// values integer
      L     #EventObject_25; // event-Nr
      T     "SSA_LOG_Value_Queue".Input.Para_0010;
      L     2; // object-state going
      T     "SSA_LOG_Value_Queue".Input.Para_0011;
      L     0; // number additional param
      T     "SSA_LOG_Value_Queue".Input.Para_0012;
// cont log-messages
      L     "SSA_LOG_Value_Queue".Input.Para_0099; // message counter
      L     1;
      +I    ;
      T     "SSA_LOG_Value_Queue".Input.Para_0099; // message counter

// Transform Basic Time to Local Time
//      CALL  "BT_LT"
//       BT     :="DB Prozesszeit".Arbeitsbereich.dt1
//       WS_DAT :="RegelDB"
//       RET_VAL:=MW218
//       LT     :="RegelDB".LocalTime
// put timestamp into message
      CALL "SYS_Copy_DBtoDB" (
           DBSource                 := 1013,
           ByteSource               := 18,
           DBDest                   := 1005,
           ByteDest                 := 462,
           NoOfByte                 := 8,
           Fault                    := M    210.0);
///
      CALL "SSA_MH_LogEntry_ActValue" (
           DBNumber                 := 1005);

E060: NOP   0;
///
// Ereignis 26  Kommt
      U     #EREIGNISBIT_26;
      FP    #Ereignis_26.FP_Kommt;
      SPBN  E061;
// header
      L     #MessageType;
      T     "SSA_LOG_Value_Queue".Input.Header.SecType; // type
      L     #MessageFormat;
      T     "SSA_LOG_Value_Queue".Input.Header.Format; // format
      L     #JobNumber;
      T     "SSA_LOG_Value_Queue".Input.Para_0005;
      L     #processMinute;
      T     "SSA_LOG_Value_Queue".Input.Para_0007;
      L     #StepNumber;
      T     "SSA_LOG_Value_Queue".Input.Para_0008;
      L     #StepTimeMin;
      T     "SSA_LOG_Value_Queue".Input.Para_0009;

// values integer
      L     #EventObject_26; // event-Nr
      T     "SSA_LOG_Value_Queue".Input.Para_0010;
      L     1; // object-state coming
      T     "SSA_LOG_Value_Queue".Input.Para_0011;
      L     0; // number additional param
      T     "SSA_LOG_Value_Queue".Input.Para_0012;
// cont log-messages
      L     "SSA_LOG_Value_Queue".Input.Para_0099; // message counter
      L     1;
      +I    ;
      T     "SSA_LOG_Value_Queue".Input.Para_0099; // message counter

// Transform Basic Time to Local Time
//      CALL  "BT_LT"
//       BT     :="DB Prozesszeit".Arbeitsbereich.dt1
//       WS_DAT :="RegelDB"
//       RET_VAL:=MW218
//       LT     :="RegelDB".LocalTime
// put timestamp into message
      CALL "SYS_Copy_DBtoDB" (
           DBSource                 := 1013,
           ByteSource               := 18,
           DBDest                   := 1005,
           ByteDest                 := 462,
           NoOfByte                 := 8,
           Fault                    := M    210.0);
///
      CALL "SSA_MH_LogEntry_ActValue" (
           DBNumber                 := 1005);

E061: NOP   0;
///
// Ereignis 26  Geht
      U     #EREIGNISBIT_26;
      FN    #Ereignis_26.FN_Geht;
      SPBN  E062;
// header
      L     #MessageType;
      T     "SSA_LOG_Value_Queue".Input.Header.SecType; // type
      L     #MessageFormat;
      T     "SSA_LOG_Value_Queue".Input.Header.Format; // format
      L     #JobNumber;
      T     "SSA_LOG_Value_Queue".Input.Para_0005;
      L     #processMinute;
      T     "SSA_LOG_Value_Queue".Input.Para_0007;
      L     #StepNumber;
      T     "SSA_LOG_Value_Queue".Input.Para_0008;
      L     #StepTimeMin;
      T     "SSA_LOG_Value_Queue".Input.Para_0009;

// values integer
      L     #EventObject_26; // event-Nr
      T     "SSA_LOG_Value_Queue".Input.Para_0010;
      L     2; // object-state going
      T     "SSA_LOG_Value_Queue".Input.Para_0011;
      L     0; // number additional param
      T     "SSA_LOG_Value_Queue".Input.Para_0012;
// cont log-messages
      L     "SSA_LOG_Value_Queue".Input.Para_0099; // message counter
      L     1;
      +I    ;
      T     "SSA_LOG_Value_Queue".Input.Para_0099; // message counter

// Transform Basic Time to Local Time
//      CALL  "BT_LT"
//       BT     :="DB Prozesszeit".Arbeitsbereich.dt1
//       WS_DAT :="RegelDB"
//       RET_VAL:=MW218
//       LT     :="RegelDB".LocalTime
// put timestamp into message
      CALL "SYS_Copy_DBtoDB" (
           DBSource                 := 1013,
           ByteSource               := 18,
           DBDest                   := 1005,
           ByteDest                 := 462,
           NoOfByte                 := 8,
           Fault                    := M    210.0);
///
      CALL "SSA_MH_LogEntry_ActValue" (
           DBNumber                 := 1005);

E062: NOP   0;
///
// Ereignis 27  Kommt
      U     #EREIGNISBIT_27;
      FP    #Ereignis_27.FP_Kommt;
      SPBN  E063;
/// header
      L     #MessageType;
      T     "SSA_LOG_Value_Queue".Input.Header.SecType; // type
      L     #MessageFormat;
      T     "SSA_LOG_Value_Queue".Input.Header.Format; // format
      L     #JobNumber;
      T     "SSA_LOG_Value_Queue".Input.Para_0005;
      L     #processMinute;
      T     "SSA_LOG_Value_Queue".Input.Para_0007;
      L     #StepNumber;
      T     "SSA_LOG_Value_Queue".Input.Para_0008;
      L     #StepTimeMin;
      T     "SSA_LOG_Value_Queue".Input.Para_0009;

// values integer
      L     #EventObject_27; // event-Nr
      T     "SSA_LOG_Value_Queue".Input.Para_0010;
      L     1; // object-state coming
      T     "SSA_LOG_Value_Queue".Input.Para_0011;
      L     0; // number additional param
      T     "SSA_LOG_Value_Queue".Input.Para_0012;
// cont log-messages
      L     "SSA_LOG_Value_Queue".Input.Para_0099; // message counter
      L     1;
      +I    ;
      T     "SSA_LOG_Value_Queue".Input.Para_0099; // message counter

// Transform Basic Time to Local Time
//      CALL  "BT_LT"
//       BT     :="DB Prozesszeit".Arbeitsbereich.dt1
//       WS_DAT :="RegelDB"
//       RET_VAL:=MW218
//       LT     :="RegelDB".LocalTime
// put timestamp into message
      CALL "SYS_Copy_DBtoDB" (
           DBSource                 := 1013,
           ByteSource               := 18,
           DBDest                   := 1005,
           ByteDest                 := 462,
           NoOfByte                 := 8,
           Fault                    := M    210.0);
///
      CALL "SSA_MH_LogEntry_ActValue" (
           DBNumber                 := 1005);

E063: NOP   0;
///
// Ereignis 27  Geht
      U     #EREIGNISBIT_27;
      FN    #Ereignis_27.FN_Geht;
      SPBN  E064;
// header
      L     #MessageType;
      T     "SSA_LOG_Value_Queue".Input.Header.SecType; // type
      L     #MessageFormat;
      T     "SSA_LOG_Value_Queue".Input.Header.Format; // format
      L     #JobNumber;
      T     "SSA_LOG_Value_Queue".Input.Para_0005;
      L     #processMinute;
      T     "SSA_LOG_Value_Queue".Input.Para_0007;
      L     #StepNumber;
      T     "SSA_LOG_Value_Queue".Input.Para_0008;
      L     #StepTimeMin;
      T     "SSA_LOG_Value_Queue".Input.Para_0009;

// values integer
      L     #EventObject_27; // event-Nr
      T     "SSA_LOG_Value_Queue".Input.Para_0010;
      L     2; // object-state going
      T     "SSA_LOG_Value_Queue".Input.Para_0011;
      L     0; // number additional param
      T     "SSA_LOG_Value_Queue".Input.Para_0012;
// cont log-messages
      L     "SSA_LOG_Value_Queue".Input.Para_0099; // message counter
      L     1;
      +I    ;
      T     "SSA_LOG_Value_Queue".Input.Para_0099; // message counter

// Transform Basic Time to Local Time
//      CALL  "BT_LT"
//       BT     :="DB Prozesszeit".Arbeitsbereich.dt1
//       WS_DAT :="RegelDB"
//       RET_VAL:=MW218
//       LT     :="RegelDB".LocalTime
// put timestamp into message
      CALL "SYS_Copy_DBtoDB" (
           DBSource                 := 1013,
           ByteSource               := 18,
           DBDest                   := 1005,
           ByteDest                 := 462,
           NoOfByte                 := 8,
           Fault                    := M    210.0);
///
      CALL "SSA_MH_LogEntry_ActValue" (
           DBNumber                 := 1005);

E064: NOP   0;
///
// Ereignis 28  Kommt
      U     #EREIGNISBIT_28;
      FP    #Ereignis_28.FP_Kommt;
      SPBN  E065;
// header
      L     #MessageType;
      T     "SSA_LOG_Value_Queue".Input.Header.SecType; // type
      L     #MessageFormat;
      T     "SSA_LOG_Value_Queue".Input.Header.Format; // format
      L     #JobNumber;
      T     "SSA_LOG_Value_Queue".Input.Para_0005;
      L     #processMinute;
      T     "SSA_LOG_Value_Queue".Input.Para_0007;
      L     #StepNumber;
      T     "SSA_LOG_Value_Queue".Input.Para_0008;
      L     #StepTimeMin;
      T     "SSA_LOG_Value_Queue".Input.Para_0009;

// values integer
      L     #EventObject_28; // event-Nr
      T     "SSA_LOG_Value_Queue".Input.Para_0010;
      L     1; // object-state coming
      T     "SSA_LOG_Value_Queue".Input.Para_0011;
      L     0; // number additional param
      T     "SSA_LOG_Value_Queue".Input.Para_0012;
// cont log-messages
      L     "SSA_LOG_Value_Queue".Input.Para_0099; // message counter
      L     1;
      +I    ;
      T     "SSA_LOG_Value_Queue".Input.Para_0099; // message counter

// Transform Basic Time to Local Time
//      CALL  "BT_LT"
//       BT     :="DB Prozesszeit".Arbeitsbereich.dt1
//       WS_DAT :="RegelDB"
//       RET_VAL:=MW218
//       LT     :="RegelDB".LocalTime
// put timestamp into message
      CALL "SYS_Copy_DBtoDB" (
           DBSource                 := 1013,
           ByteSource               := 18,
           DBDest                   := 1005,
           ByteDest                 := 462,
           NoOfByte                 := 8,
           Fault                    := M    210.0);
///
      CALL "SSA_MH_LogEntry_ActValue" (
           DBNumber                 := 1005);

E065: NOP   0;
///
// Ereignis 28  Geht
      U     #EREIGNISBIT_28;
      FN    #Ereignis_28.FN_Geht;
      SPBN  E066;
// header
      L     #MessageType;
      T     "SSA_LOG_Value_Queue".Input.Header.SecType; // type
      L     #MessageFormat;
      T     "SSA_LOG_Value_Queue".Input.Header.Format; // format
      L     #JobNumber;
      T     "SSA_LOG_Value_Queue".Input.Para_0005;
      L     #processMinute;
      T     "SSA_LOG_Value_Queue".Input.Para_0007;
      L     #StepNumber;
      T     "SSA_LOG_Value_Queue".Input.Para_0008;
      L     #StepTimeMin;
      T     "SSA_LOG_Value_Queue".Input.Para_0009;

// values integer
      L     #EventObject_28; // event-Nr
      T     "SSA_LOG_Value_Queue".Input.Para_0010;
      L     2; // object-state going
      T     "SSA_LOG_Value_Queue".Input.Para_0011;
      L     0; // number additional param
      T     "SSA_LOG_Value_Queue".Input.Para_0012;
// cont log-messages
      L     "SSA_LOG_Value_Queue".Input.Para_0099; // message counter
      L     1;
      +I    ;
      T     "SSA_LOG_Value_Queue".Input.Para_0099; // message counter

// Transform Basic Time to Local Time
//      CALL  "BT_LT"
//       BT     :="DB Prozesszeit".Arbeitsbereich.dt1
//       WS_DAT :="RegelDB"
//       RET_VAL:=MW218
//       LT     :="RegelDB".LocalTime
// put timestamp into message
      CALL "SYS_Copy_DBtoDB" (
           DBSource                 := 1013,
           ByteSource               := 18,
           DBDest                   := 1005,
           ByteDest                 := 462,
           NoOfByte                 := 8,
           Fault                    := M    210.0);
///
      CALL "SSA_MH_LogEntry_ActValue" (
           DBNumber                 := 1005);

E066: NOP   0;
///
// Ereignis 29  Kommt
      U     #EREIGNISBIT_29;
      FP    #Ereignis_29.FP_Kommt;
      SPBN  E067;
// header
      L     #MessageType;
      T     "SSA_LOG_Value_Queue".Input.Header.SecType; // type
      L     #MessageFormat;
      T     "SSA_LOG_Value_Queue".Input.Header.Format; // format
      L     #JobNumber;
      T     "SSA_LOG_Value_Queue".Input.Para_0005;
      L     #processMinute;
      T     "SSA_LOG_Value_Queue".Input.Para_0007;
      L     #StepNumber;
      T     "SSA_LOG_Value_Queue".Input.Para_0008;
      L     #StepTimeMin;
      T     "SSA_LOG_Value_Queue".Input.Para_0009;

// values integer
      L     #EventObject_29; // event-Nr
      T     "SSA_LOG_Value_Queue".Input.Para_0010;
      L     1; // object-state coming
      T     "SSA_LOG_Value_Queue".Input.Para_0011;
      L     0; // number additional param
      T     "SSA_LOG_Value_Queue".Input.Para_0012;
// cont log-messages
      L     "SSA_LOG_Value_Queue".Input.Para_0099; // message counter
      L     1;
      +I    ;
      T     "SSA_LOG_Value_Queue".Input.Para_0099; // message counter

// Transform Basic Time to Local Time
//      CALL  "BT_LT"
//       BT     :="DB Prozesszeit".Arbeitsbereich.dt1
//       WS_DAT :="RegelDB"
//       RET_VAL:=MW218
//       LT     :="RegelDB".LocalTime
// put timestamp into message
      CALL "SYS_Copy_DBtoDB" (
           DBSource                 := 1013,
           ByteSource               := 18,
           DBDest                   := 1005,
           ByteDest                 := 462,
           NoOfByte                 := 8,
           Fault                    := M    210.0);
///
      CALL "SSA_MH_LogEntry_ActValue" (
           DBNumber                 := 1005);

E067: NOP   0;
///
// Ereignis 29  Geht
      U     #EREIGNISBIT_29;
      FN    #Ereignis_29.FN_Geht;
      SPBN  E068;
// header
      L     #MessageType;
      T     "SSA_LOG_Value_Queue".Input.Header.SecType; // type
      L     #MessageFormat;
      T     "SSA_LOG_Value_Queue".Input.Header.Format; // format
      L     #JobNumber;
      T     "SSA_LOG_Value_Queue".Input.Para_0005;
      L     #processMinute;
      T     "SSA_LOG_Value_Queue".Input.Para_0007;
      L     #StepNumber;
      T     "SSA_LOG_Value_Queue".Input.Para_0008;
      L     #StepTimeMin;
      T     "SSA_LOG_Value_Queue".Input.Para_0009;

// values integer
      L     #EventObject_29; // event-Nr
      T     "SSA_LOG_Value_Queue".Input.Para_0010;
      L     2; // object-state going
      T     "SSA_LOG_Value_Queue".Input.Para_0011;
      L     0; // number additional param
      T     "SSA_LOG_Value_Queue".Input.Para_0012;
// cont log-messages
      L     "SSA_LOG_Value_Queue".Input.Para_0099; // message counter
      L     1;
      +I    ;
      T     "SSA_LOG_Value_Queue".Input.Para_0099; // message counter

// Transform Basic Time to Local Time
//      CALL  "BT_LT"
//       BT     :="DB Prozesszeit".Arbeitsbereich.dt1
//       WS_DAT :="RegelDB"
//       RET_VAL:=MW218
//       LT     :="RegelDB".LocalTime
// put timestamp into message
      CALL "SYS_Copy_DBtoDB" (
           DBSource                 := 1013,
           ByteSource               := 18,
           DBDest                   := 1005,
           ByteDest                 := 462,
           NoOfByte                 := 8,
           Fault                    := M    210.0);
///
      CALL "SSA_MH_LogEntry_ActValue" (
           DBNumber                 := 1005);

E068: NOP   0;
///
// Ereignis 30  Kommt
      U     #EREIGNISBIT_30;
      FP    #Ereignis_30.FP_Kommt;
      SPBN  E069;
// header
      L     #MessageType;
      T     "SSA_LOG_Value_Queue".Input.Header.SecType; // type
      L     #MessageFormat;
      T     "SSA_LOG_Value_Queue".Input.Header.Format; // format
      L     #JobNumber;
      T     "SSA_LOG_Value_Queue".Input.Para_0005;
      L     #processMinute;
      T     "SSA_LOG_Value_Queue".Input.Para_0007;
      L     #StepNumber;
      T     "SSA_LOG_Value_Queue".Input.Para_0008;
      L     #StepTimeMin;
      T     "SSA_LOG_Value_Queue".Input.Para_0009;

// values integer
      L     #EventObject_30; // event-Nr
      T     "SSA_LOG_Value_Queue".Input.Para_0010;
      L     1; // object-state coming
      T     "SSA_LOG_Value_Queue".Input.Para_0011;
      L     0; // number additional param
      T     "SSA_LOG_Value_Queue".Input.Para_0012;
// cont log-messages
      L     "SSA_LOG_Value_Queue".Input.Para_0099; // message counter
      L     1;
      +I    ;
      T     "SSA_LOG_Value_Queue".Input.Para_0099; // message counter

// Transform Basic Time to Local Time
//      CALL  "BT_LT"
//       BT     :="DB Prozesszeit".Arbeitsbereich.dt1
//       WS_DAT :="RegelDB"
//       RET_VAL:=MW218
//       LT     :="RegelDB".LocalTime
// put timestamp into message
      CALL "SYS_Copy_DBtoDB" (
           DBSource                 := 1013,
           ByteSource               := 18,
           DBDest                   := 1005,
           ByteDest                 := 462,
           NoOfByte                 := 8,
           Fault                    := M    210.0);
///
      CALL "SSA_MH_LogEntry_ActValue" (
           DBNumber                 := 1005);

E069: NOP   0;
///
// Ereignis 30  Geht
      U     #EREIGNISBIT_30;
      FN    #Ereignis_30.FN_Geht;
      SPBN  E070;
// header
      L     #MessageType;
      T     "SSA_LOG_Value_Queue".Input.Header.SecType; // type
      L     #MessageFormat;
      T     "SSA_LOG_Value_Queue".Input.Header.Format; // format
      L     #JobNumber;
      T     "SSA_LOG_Value_Queue".Input.Para_0005;
      L     #processMinute;
      T     "SSA_LOG_Value_Queue".Input.Para_0007;
      L     #StepNumber;
      T     "SSA_LOG_Value_Queue".Input.Para_0008;
      L     #StepTimeMin;
      T     "SSA_LOG_Value_Queue".Input.Para_0009;

// values integer
      L     #EventObject_30; // event-Nr
      T     "SSA_LOG_Value_Queue".Input.Para_0010;
      L     2; // object-state going
      T     "SSA_LOG_Value_Queue".Input.Para_0011;
      L     0; // number additional param
      T     "SSA_LOG_Value_Queue".Input.Para_0012;
// cont log-messages
      L     "SSA_LOG_Value_Queue".Input.Para_0099; // message counter
      L     1;
      +I    ;
      T     "SSA_LOG_Value_Queue".Input.Para_0099; // message counter

// Transform Basic Time to Local Time
//      CALL  "BT_LT"
//       BT     :="DB Prozesszeit".Arbeitsbereich.dt1
//       WS_DAT :="RegelDB"
//       RET_VAL:=MW218
//       LT     :="RegelDB".LocalTime
// put timestamp into message
      CALL "SYS_Copy_DBtoDB" (
           DBSource                 := 1013,
           ByteSource               := 18,
           DBDest                   := 1005,
           ByteDest                 := 462,
           NoOfByte                 := 8,
           Fault                    := M    210.0);
///
      CALL "SSA_MH_LogEntry_ActValue" (
           DBNumber                 := 1005);

E070: NOP   0;
///

NETWORK
TITLE =create events for batchprotokoll
//event Nr. 121 - 130 are  events in job-protocol
///
// Ereignis 31  Kommt
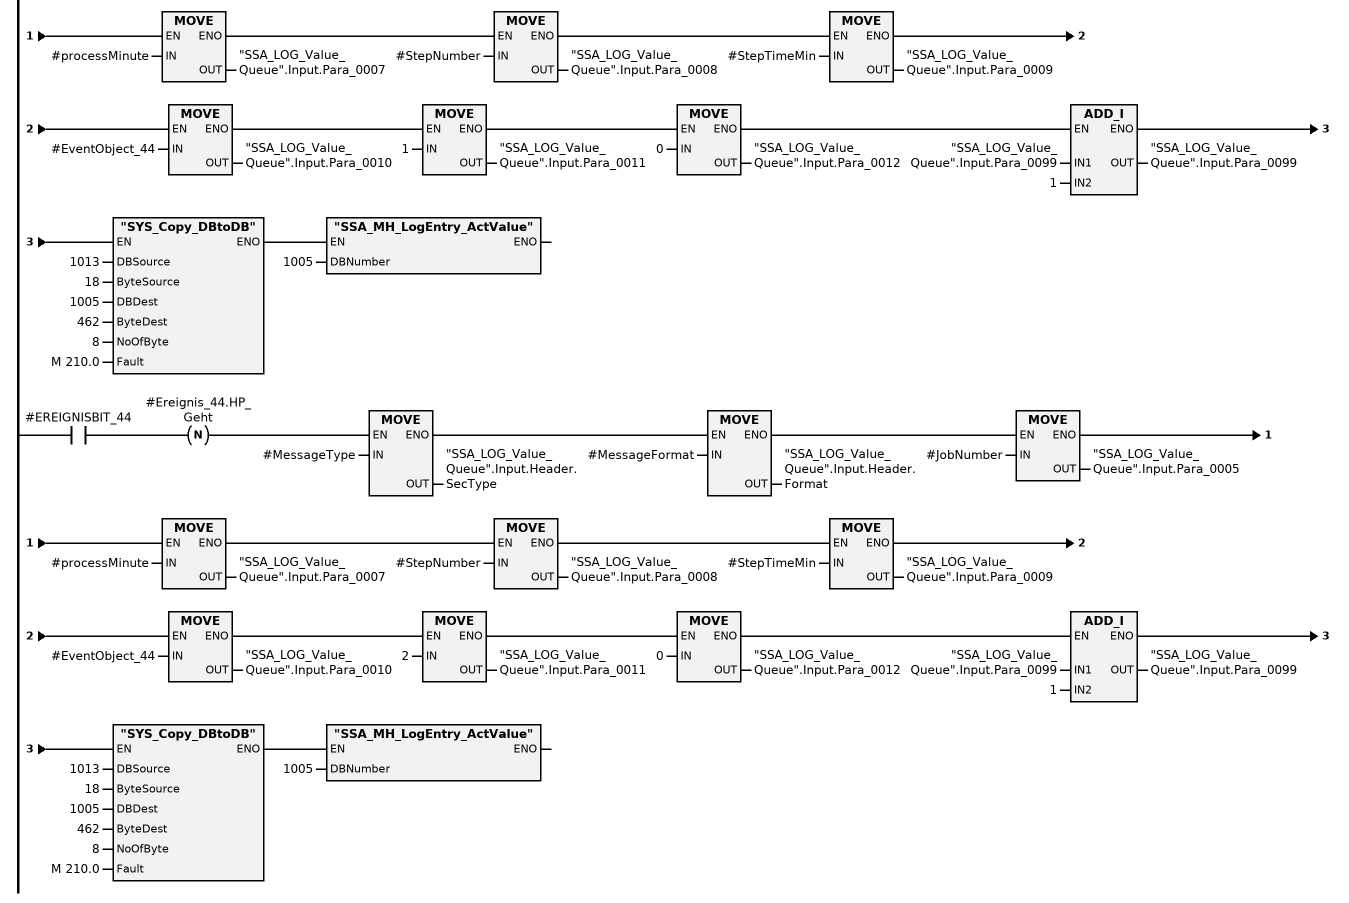
      U     #EREIGNISBIT_31;
      FP    #Ereignis_31.FP_Kommt;
      SPBN  E071;
// header
      L     #MessageType;
      T     "SSA_LOG_Value_Queue".Input.Header.SecType; // type
      L     #MessageFormat;
      T     "SSA_LOG_Value_Queue".Input.Header.Format; // format
      L     #JobNumber;
      T     "SSA_LOG_Value_Queue".Input.Para_0005;
      L     #processMinute;
      T     "SSA_LOG_Value_Queue".Input.Para_0007;
      L     #StepNumber;
      T     "SSA_LOG_Value_Queue".Input.Para_0008;
      L     #StepTimeMin;
      T     "SSA_LOG_Value_Queue".Input.Para_0009;

// values integer
      L     #EventObject_31; // event-Nr
      T     "SSA_LOG_Value_Queue".Input.Para_0010;
      L     1; // object-state coming
      T     "SSA_LOG_Value_Queue".Input.Para_0011;
      L     0; // number additional param
      T     "SSA_LOG_Value_Queue".Input.Para_0012;
// cont log-messages
      L     "SSA_LOG_Value_Queue".Input.Para_0099; // message counter
      L     1;
      +I    ;
      T     "SSA_LOG_Value_Queue".Input.Para_0099; // message counter

// Transform Basic Time to Local Time
//      CALL  "BT_LT"
//       BT     :="DB Prozesszeit".Arbeitsbereich.dt1
//       WS_DAT :="RegelDB"
//       RET_VAL:=MW218
//       LT     :="RegelDB".LocalTime
// put timestamp into message
      CALL "SYS_Copy_DBtoDB" (
           DBSource                 := 1013,
           ByteSource               := 18,
           DBDest                   := 1005,
           ByteDest                 := 462,
           NoOfByte                 := 8,
           Fault                    := M    210.0);
///
      CALL "SSA_MH_LogEntry_ActValue" (
           DBNumber                 := 1005);
E071: NOP   0;
///
// Ereignis 31  Geht
      U     #EREIGNISBIT_31;
      FN    #Ereignis_31.FN_Geht;
      SPBN  E072;
// header
      L     #MessageType;
      T     "SSA_LOG_Value_Queue".Input.Header.SecType; // type
      L     #MessageFormat;
      T     "SSA_LOG_Value_Queue".Input.Header.Format; // format
      L     #JobNumber;
      T     "SSA_LOG_Value_Queue".Input.Para_0005;
      L     #processMinute;
      T     "SSA_LOG_Value_Queue".Input.Para_0007;
      L     #StepNumber;
      T     "SSA_LOG_Value_Queue".Input.Para_0008;
      L     #StepTimeMin;
      T     "SSA_LOG_Value_Queue".Input.Para_0009;

// values integer
      L     #EventObject_31; // event-Nr
      T     "SSA_LOG_Value_Queue".Input.Para_0010;
      L     2; // object-state going
      T     "SSA_LOG_Value_Queue".Input.Para_0011;
      L     0; // number additional param
      T     "SSA_LOG_Value_Queue".Input.Para_0012;
// cont log-messages
      L     "SSA_LOG_Value_Queue".Input.Para_0099; // message counter
      L     1;
      +I    ;
      T     "SSA_LOG_Value_Queue".Input.Para_0099; // message counter

// Transform Basic Time to Local Time
//      CALL  "BT_LT"
//       BT     :="DB Prozesszeit".Arbeitsbereich.dt1
//       WS_DAT :="RegelDB"
//       RET_VAL:=MW218
//       LT     :="RegelDB".LocalTime
// put timestamp into message
      CALL "SYS_Copy_DBtoDB" (
           DBSource                 := 1013,
           ByteSource               := 18,
           DBDest                   := 1005,
           ByteDest                 := 462,
           NoOfByte                 := 8,
           Fault                    := M    210.0);
///
      CALL "SSA_MH_LogEntry_ActValue" (
           DBNumber                 := 1005);

E072: NOP   0;
///
// Ereignis 32  Kommt
      U     #EREIGNISBIT_32;
      FP    #Ereignis_32.FP_Kommt;
      SPBN  E073;
// header
      L     #MessageType;
      T     "SSA_LOG_Value_Queue".Input.Header.SecType; // type
      L     #MessageFormat;
      T     "SSA_LOG_Value_Queue".Input.Header.Format; // format
      L     #JobNumber;
      T     "SSA_LOG_Value_Queue".Input.Para_0005;
      L     #processMinute;
      T     "SSA_LOG_Value_Queue".Input.Para_0007;
      L     #StepNumber;
      T     "SSA_LOG_Value_Queue".Input.Para_0008;
      L     #StepTimeMin;
      T     "SSA_LOG_Value_Queue".Input.Para_0009;

// values integer
      L     #EventObject_32; // event-Nr
      T     "SSA_LOG_Value_Queue".Input.Para_0010;
      L     1; // object-state coming
      T     "SSA_LOG_Value_Queue".Input.Para_0011;
      L     0; // number additional param
      T     "SSA_LOG_Value_Queue".Input.Para_0012;
// cont log-messages
      L     "SSA_LOG_Value_Queue".Input.Para_0099; // message counter
      L     1;
      +I    ;
      T     "SSA_LOG_Value_Queue".Input.Para_0099; // message counter

// Transform Basic Time to Local Time
//      CALL  "BT_LT"
//       BT     :="DB Prozesszeit".Arbeitsbereich.dt1
//       WS_DAT :="RegelDB"
//       RET_VAL:=MW218
//       LT     :="RegelDB".LocalTime
// put timestamp into message
      CALL "SYS_Copy_DBtoDB" (
           DBSource                 := 1013,
           ByteSource               := 18,
           DBDest                   := 1005,
           ByteDest                 := 462,
           NoOfByte                 := 8,
           Fault                    := M    210.0);
///
      CALL "SSA_MH_LogEntry_ActValue" (
           DBNumber                 := 1005);

E073: NOP   0;
///
// Ereignis 32  Geht
      U     #EREIGNISBIT_32;
      FN    #Ereignis_32.FN_Geht;
      SPBN  E074;
// header
      L     #MessageType;
      T     "SSA_LOG_Value_Queue".Input.Header.SecType; // type
      L     #MessageFormat;
      T     "SSA_LOG_Value_Queue".Input.Header.Format; // format
      L     #JobNumber;
      T     "SSA_LOG_Value_Queue".Input.Para_0005;
      L     #processMinute;
      T     "SSA_LOG_Value_Queue".Input.Para_0007;
      L     #StepNumber;
      T     "SSA_LOG_Value_Queue".Input.Para_0008;
      L     #StepTimeMin;
      T     "SSA_LOG_Value_Queue".Input.Para_0009;

// values integer
      L     #EventObject_32; // event-Nr
      T     "SSA_LOG_Value_Queue".Input.Para_0010;
      L     2; // object-state going
      T     "SSA_LOG_Value_Queue".Input.Para_0011;
      L     0; // number additional param
      T     "SSA_LOG_Value_Queue".Input.Para_0012;
// cont log-messages
      L     "SSA_LOG_Value_Queue".Input.Para_0099; // message counter
      L     1;
      +I    ;
      T     "SSA_LOG_Value_Queue".Input.Para_0099; // message counter

// Transform Basic Time to Local Time
//      CALL  "BT_LT"
//       BT     :="DB Prozesszeit".Arbeitsbereich.dt1
//       WS_DAT :="RegelDB"
//       RET_VAL:=MW218
//       LT     :="RegelDB".LocalTime
// put timestamp into message
      CALL "SYS_Copy_DBtoDB" (
           DBSource                 := 1013,
           ByteSource               := 18,
           DBDest                   := 1005,
           ByteDest                 := 462,
           NoOfByte                 := 8,
           Fault                    := M    210.0);
///
      CALL "SSA_MH_LogEntry_ActValue" (
           DBNumber                 := 1005);

E074: NOP   0;
///
// Ereignis 33  Kommt
      U     #EREIGNISBIT_33;
      FP    #Ereignis_33.FP_Kommt;
      SPBN  E075;
// header
      L     #MessageType;
      T     "SSA_LOG_Value_Queue".Input.Header.SecType; // type
      L     #MessageFormat;
      T     "SSA_LOG_Value_Queue".Input.Header.Format; // format
      L     #JobNumber;
      T     "SSA_LOG_Value_Queue".Input.Para_0005;
      L     #processMinute;
      T     "SSA_LOG_Value_Queue".Input.Para_0007;
      L     #StepNumber;
      T     "SSA_LOG_Value_Queue".Input.Para_0008;
      L     #StepTimeMin;
      T     "SSA_LOG_Value_Queue".Input.Para_0009;

// values integer
      L     #EventObject_33; // event-Nr
      T     "SSA_LOG_Value_Queue".Input.Para_0010;
      L     1; // object-state coming
      T     "SSA_LOG_Value_Queue".Input.Para_0011;
      L     0; // number additional param
      T     "SSA_LOG_Value_Queue".Input.Para_0012;
// cont log-messages
      L     "SSA_LOG_Value_Queue".Input.Para_0099; // message counter
      L     1;
      +I    ;
      T     "SSA_LOG_Value_Queue".Input.Para_0099; // message counter

// Transform Basic Time to Local Time
//      CALL  "BT_LT"
//       BT     :="DB Prozesszeit".Arbeitsbereich.dt1
//       WS_DAT :="RegelDB"
//       RET_VAL:=MW218
//       LT     :="RegelDB".LocalTime
// put timestamp into message
      CALL "SYS_Copy_DBtoDB" (
           DBSource                 := 1013,
           ByteSource               := 18,
           DBDest                   := 1005,
           ByteDest                 := 462,
           NoOfByte                 := 8,
           Fault                    := M    210.0);
///
      CALL "SSA_MH_LogEntry_ActValue" (
           DBNumber                 := 1005);

E075: NOP   0;
///
// Ereignis 33  Geht
      U     #EREIGNISBIT_33;
      FN    #Ereignis_33.FN_Geht;
      SPBN  E076;
// header
      L     #MessageType;
      T     "SSA_LOG_Value_Queue".Input.Header.SecType; // type
      L     #MessageFormat;
      T     "SSA_LOG_Value_Queue".Input.Header.Format; // format
      L     #JobNumber;
      T     "SSA_LOG_Value_Queue".Input.Para_0005;
      L     #processMinute;
      T     "SSA_LOG_Value_Queue".Input.Para_0007;
      L     #StepNumber;
      T     "SSA_LOG_Value_Queue".Input.Para_0008;
      L     #StepTimeMin;
      T     "SSA_LOG_Value_Queue".Input.Para_0009;

// values integer
      L     #EventObject_33; // event-Nr
      T     "SSA_LOG_Value_Queue".Input.Para_0010;
      L     2; // object-state going
      T     "SSA_LOG_Value_Queue".Input.Para_0011;
      L     0; // number additional param
      T     "SSA_LOG_Value_Queue".Input.Para_0012;
// cont log-messages
      L     "SSA_LOG_Value_Queue".Input.Para_0099; // message counter
      L     1;
      +I    ;
      T     "SSA_LOG_Value_Queue".Input.Para_0099; // message counter

// Transform Basic Time to Local Time
//      CALL  "BT_LT"
//       BT     :="DB Prozesszeit".Arbeitsbereich.dt1
//       WS_DAT :="RegelDB"
//       RET_VAL:=MW218
//       LT     :="RegelDB".LocalTime
// put timestamp into message
      CALL "SYS_Copy_DBtoDB" (
           DBSource                 := 1013,
           ByteSource               := 18,
           DBDest                   := 1005,
           ByteDest                 := 462,
           NoOfByte                 := 8,
           Fault                    := M    210.0);
///
      CALL "SSA_MH_LogEntry_ActValue" (
           DBNumber                 := 1005);

E076: NOP   0;
///
// Ereignis 34  Kommt
      U     #EREIGNISBIT_34;
      FP    #Ereignis_34.FP_Kommt;
      SPBN  E077;
// header
      L     #MessageType;
      T     "SSA_LOG_Value_Queue".Input.Header.SecType; // type
      L     #MessageFormat;
      T     "SSA_LOG_Value_Queue".Input.Header.Format; // format
      L     #JobNumber;
      T     "SSA_LOG_Value_Queue".Input.Para_0005;
      L     #processMinute;
      T     "SSA_LOG_Value_Queue".Input.Para_0007;
      L     #StepNumber;
      T     "SSA_LOG_Value_Queue".Input.Para_0008;
      L     #StepTimeMin;
      T     "SSA_LOG_Value_Queue".Input.Para_0009;

// values integer
      L     #EventObject_34; // event-Nr
      T     "SSA_LOG_Value_Queue".Input.Para_0010;
      L     1; // object-state coming
      T     "SSA_LOG_Value_Queue".Input.Para_0011;
      L     0; // number additional param
      T     "SSA_LOG_Value_Queue".Input.Para_0012;
// cont log-messages
      L     "SSA_LOG_Value_Queue".Input.Para_0099; // message counter
      L     1;
      +I    ;
      T     "SSA_LOG_Value_Queue".Input.Para_0099; // message counter

// Transform Basic Time to Local Time
//      CALL  "BT_LT"
//       BT     :="DB Prozesszeit".Arbeitsbereich.dt1
//       WS_DAT :="RegelDB"
//       RET_VAL:=MW218
//       LT     :="RegelDB".LocalTime
// put timestamp into message
      CALL "SYS_Copy_DBtoDB" (
           DBSource                 := 1013,
           ByteSource               := 18,
           DBDest                   := 1005,
           ByteDest                 := 462,
           NoOfByte                 := 8,
           Fault                    := M    210.0);
///
      CALL "SSA_MH_LogEntry_ActValue" (
           DBNumber                 := 1005);

E077: NOP   0;
///
// Ereignis 34  Geht
      U     #EREIGNISBIT_34;
      FN    #Ereignis_34.FN_Geht;
      SPBN  E078;
// header
      L     #MessageType;
      T     "SSA_LOG_Value_Queue".Input.Header.SecType; // type
      L     #MessageFormat;
      T     "SSA_LOG_Value_Queue".Input.Header.Format; // format
      L     #JobNumber;
      T     "SSA_LOG_Value_Queue".Input.Para_0005;
      L     #processMinute;
      T     "SSA_LOG_Value_Queue".Input.Para_0007;
      L     #StepNumber;
      T     "SSA_LOG_Value_Queue".Input.Para_0008;
      L     #StepTimeMin;
      T     "SSA_LOG_Value_Queue".Input.Para_0009;

// values integer
      L     #EventObject_34; // event-Nr
      T     "SSA_LOG_Value_Queue".Input.Para_0010;
      L     2; // object-state going
      T     "SSA_LOG_Value_Queue".Input.Para_0011;
      L     0; // number additional param
      T     "SSA_LOG_Value_Queue".Input.Para_0012;
// cont log-messages
      L     "SSA_LOG_Value_Queue".Input.Para_0099; // message counter
      L     1;
      +I    ;
      T     "SSA_LOG_Value_Queue".Input.Para_0099; // message counter

// Transform Basic Time to Local Time
//      CALL  "BT_LT"
//       BT     :="DB Prozesszeit".Arbeitsbereich.dt1
//       WS_DAT :="RegelDB"
//       RET_VAL:=MW218
//       LT     :="RegelDB".LocalTime
// put timestamp into message
      CALL "SYS_Copy_DBtoDB" (
           DBSource                 := 1013,
           ByteSource               := 18,
           DBDest                   := 1005,
           ByteDest                 := 462,
           NoOfByte                 := 8,
           Fault                    := M    210.0);
///
      CALL "SSA_MH_LogEntry_ActValue" (
           DBNumber                 := 1005);

E078: NOP   0;
///
// Ereignis 35  Kommt
      U     #EREIGNISBIT_35;
      FP    #Ereignis_35.FP_Kommt;
      SPBN  E079;
// header
      L     #MessageType;
      T     "SSA_LOG_Value_Queue".Input.Header.SecType; // type
      L     #MessageFormat;
      T     "SSA_LOG_Value_Queue".Input.Header.Format; // format
      L     #JobNumber;
      T     "SSA_LOG_Value_Queue".Input.Para_0005;
      L     #processMinute;
      T     "SSA_LOG_Value_Queue".Input.Para_0007;
      L     #StepNumber;
      T     "SSA_LOG_Value_Queue".Input.Para_0008;
      L     #StepTimeMin;
      T     "SSA_LOG_Value_Queue".Input.Para_0009;

// values integer
      L     #EventObject_35; // event-Nr
      T     "SSA_LOG_Value_Queue".Input.Para_0010;
      L     1; // object-state coming
      T     "SSA_LOG_Value_Queue".Input.Para_0011;
      L     0; // number additional param
      T     "SSA_LOG_Value_Queue".Input.Para_0012;
// cont log-messages
      L     "SSA_LOG_Value_Queue".Input.Para_0099; // message counter
      L     1;
      +I    ;
      T     "SSA_LOG_Value_Queue".Input.Para_0099; // message counter

// Transform Basic Time to Local Time
//      CALL  "BT_LT"
//       BT     :="DB Prozesszeit".Arbeitsbereich.dt1
//       WS_DAT :="RegelDB"
//       RET_VAL:=MW218
//       LT     :="RegelDB".LocalTime
// put timestamp into message
      CALL "SYS_Copy_DBtoDB" (
           DBSource                 := 1013,
           ByteSource               := 18,
           DBDest                   := 1005,
           ByteDest                 := 462,
           NoOfByte                 := 8,
           Fault                    := M    210.0);
///
      CALL "SSA_MH_LogEntry_ActValue" (
           DBNumber                 := 1005);

E079: NOP   0;
///
// Ereignis 35  Geht
      U     #EREIGNISBIT_35;
      FN    #Ereignis_35.FN_Geht;
      SPBN  E080;
// header
      L     #MessageType;
      T     "SSA_LOG_Value_Queue".Input.Header.SecType; // type
      L     #MessageFormat;
      T     "SSA_LOG_Value_Queue".Input.Header.Format; // format
      L     #JobNumber;
      T     "SSA_LOG_Value_Queue".Input.Para_0005;
      L     #processMinute;
      T     "SSA_LOG_Value_Queue".Input.Para_0007;
      L     #StepNumber;
      T     "SSA_LOG_Value_Queue".Input.Para_0008;
      L     #StepTimeMin;
      T     "SSA_LOG_Value_Queue".Input.Para_0009;

// values integer
      L     #EventObject_35; // event-Nr
      T     "SSA_LOG_Value_Queue".Input.Para_0010;
      L     2; // object-state going
      T     "SSA_LOG_Value_Queue".Input.Para_0011;
      L     0; // number additional param
      T     "SSA_LOG_Value_Queue".Input.Para_0012;
// cont log-messages
      L     "SSA_LOG_Value_Queue".Input.Para_0099; // message counter
      L     1;
      +I    ;
      T     "SSA_LOG_Value_Queue".Input.Para_0099; // message counter

// Transform Basic Time to Local Time
//      CALL  "BT_LT"
//       BT     :="DB Prozesszeit".Arbeitsbereich.dt1
//       WS_DAT :="RegelDB"
//       RET_VAL:=MW218
//       LT     :="RegelDB".LocalTime
// put timestamp into message
      CALL "SYS_Copy_DBtoDB" (
           DBSource                 := 1013,
           ByteSource               := 18,
           DBDest                   := 1005,
           ByteDest                 := 462,
           NoOfByte                 := 8,
           Fault                    := M    210.0);
///
      CALL "SSA_MH_LogEntry_ActValue" (
           DBNumber                 := 1005);

E080: NOP   0;
///
// Ereignis 36  Kommt
      U     #EREIGNISBIT_36;
      FP    #Ereignis_36.FP_Kommt;
      SPBN  E081;
// header
      L     #MessageType;
      T     "SSA_LOG_Value_Queue".Input.Header.SecType; // type
      L     #MessageFormat;
      T     "SSA_LOG_Value_Queue".Input.Header.Format; // format
      L     #JobNumber;
      T     "SSA_LOG_Value_Queue".Input.Para_0005;
      L     #processMinute;
      T     "SSA_LOG_Value_Queue".Input.Para_0007;
      L     #StepNumber;
      T     "SSA_LOG_Value_Queue".Input.Para_0008;
      L     #StepTimeMin;
      T     "SSA_LOG_Value_Queue".Input.Para_0009;

// values integer
      L     #EventObject_36; // event-Nr
      T     "SSA_LOG_Value_Queue".Input.Para_0010;
      L     1; // object-state coming
      T     "SSA_LOG_Value_Queue".Input.Para_0011;
      L     0; // number additional param
      T     "SSA_LOG_Value_Queue".Input.Para_0012;
// cont log-messages
      L     "SSA_LOG_Value_Queue".Input.Para_0099; // message counter
      L     1;
      +I    ;
      T     "SSA_LOG_Value_Queue".Input.Para_0099; // message counter

// Transform Basic Time to Local Time
//      CALL  "BT_LT"
//       BT     :="DB Prozesszeit".Arbeitsbereich.dt1
//       WS_DAT :="RegelDB"
//       RET_VAL:=MW218
//       LT     :="RegelDB".LocalTime
// put timestamp into message
      CALL "SYS_Copy_DBtoDB" (
           DBSource                 := 1013,
           ByteSource               := 18,
           DBDest                   := 1005,
           ByteDest                 := 462,
           NoOfByte                 := 8,
           Fault                    := M    210.0);
///
      CALL "SSA_MH_LogEntry_ActValue" (
           DBNumber                 := 1005);

E081: NOP   0;
///
// Ereignis 36  Geht
      U     #EREIGNISBIT_36;
      FN    #Ereignis_36.FN_Geht;
      SPBN  E082;
// header
      L     #MessageType;
      T     "SSA_LOG_Value_Queue".Input.Header.SecType; // type
      L     #MessageFormat;
      T     "SSA_LOG_Value_Queue".Input.Header.Format; // format
      L     #JobNumber;
      T     "SSA_LOG_Value_Queue".Input.Para_0005;
      L     #processMinute;
      T     "SSA_LOG_Value_Queue".Input.Para_0007;
      L     #StepNumber;
      T     "SSA_LOG_Value_Queue".Input.Para_0008;
      L     #StepTimeMin;
      T     "SSA_LOG_Value_Queue".Input.Para_0009;

// values integer
      L     #EventObject_36; // event-Nr
      T     "SSA_LOG_Value_Queue".Input.Para_0010;
      L     2; // object-state going
      T     "SSA_LOG_Value_Queue".Input.Para_0011;
      L     0; // number additional param
      T     "SSA_LOG_Value_Queue".Input.Para_0012;
// cont log-messages
      L     "SSA_LOG_Value_Queue".Input.Para_0099; // message counter
      L     1;
      +I    ;
      T     "SSA_LOG_Value_Queue".Input.Para_0099; // message counter

// Transform Basic Time to Local Time
//      CALL  "BT_LT"
//       BT     :="DB Prozesszeit".Arbeitsbereich.dt1
//       WS_DAT :="RegelDB"
//       RET_VAL:=MW218
//       LT     :="RegelDB".LocalTime
// put timestamp into message
      CALL "SYS_Copy_DBtoDB" (
           DBSource                 := 1013,
           ByteSource               := 18,
           DBDest                   := 1005,
           ByteDest                 := 462,
           NoOfByte                 := 8,
           Fault                    := M    210.0);
///
      CALL "SSA_MH_LogEntry_ActValue" (
           DBNumber                 := 1005);

E082: NOP   0;
///
// Ereignis 37  Kommt
      U     #EREIGNISBIT_37;
      FP    #Ereignis_37.FP_Kommt;
      SPBN  E083;
// header
      L     #MessageType;
      T     "SSA_LOG_Value_Queue".Input.Header.SecType; // type
      L     #MessageFormat;
      T     "SSA_LOG_Value_Queue".Input.Header.Format; // format
      L     #JobNumber;
      T     "SSA_LOG_Value_Queue".Input.Para_0005;
      L     #processMinute;
      T     "SSA_LOG_Value_Queue".Input.Para_0007;
      L     #StepNumber;
      T     "SSA_LOG_Value_Queue".Input.Para_0008;
      L     #StepTimeMin;
      T     "SSA_LOG_Value_Queue".Input.Para_0009;

// values integer
      L     #EventObject_37; // event-Nr
      T     "SSA_LOG_Value_Queue".Input.Para_0010;
      L     1; // object-state coming
      T     "SSA_LOG_Value_Queue".Input.Para_0011;
      L     0; // number additional param
      T     "SSA_LOG_Value_Queue".Input.Para_0012;
// cont log-messages
      L     "SSA_LOG_Value_Queue".Input.Para_0099; // message counter
      L     1;
      +I    ;
      T     "SSA_LOG_Value_Queue".Input.Para_0099; // message counter

// Transform Basic Time to Local Time
//      CALL  "BT_LT"
//       BT     :="DB Prozesszeit".Arbeitsbereich.dt1
//       WS_DAT :="RegelDB"
//       RET_VAL:=MW218
//       LT     :="RegelDB".LocalTime
// put timestamp into message
      CALL "SYS_Copy_DBtoDB" (
           DBSource                 := 1013,
           ByteSource               := 18,
           DBDest                   := 1005,
           ByteDest                 := 462,
           NoOfByte                 := 8,
           Fault                    := M    210.0);
///
      CALL "SSA_MH_LogEntry_ActValue" (
           DBNumber                 := 1005);

E083: NOP   0;
///
// Ereignis 37  Geht
      U     #EREIGNISBIT_37;
      FN    #Ereignis_37.FN_Geht;
      SPBN  E084;
// header
      L     #MessageType;
      T     "SSA_LOG_Value_Queue".Input.Header.SecType; // type
      L     #MessageFormat;
      T     "SSA_LOG_Value_Queue".Input.Header.Format; // format
      L     #JobNumber;
      T     "SSA_LOG_Value_Queue".Input.Para_0005;
      L     #processMinute;
      T     "SSA_LOG_Value_Queue".Input.Para_0007;
      L     #StepNumber;
      T     "SSA_LOG_Value_Queue".Input.Para_0008;
      L     #StepTimeMin;
      T     "SSA_LOG_Value_Queue".Input.Para_0009;

// values integer
      L     #EventObject_37; // event-Nr
      T     "SSA_LOG_Value_Queue".Input.Para_0010;
      L     2; // object-state going
      T     "SSA_LOG_Value_Queue".Input.Para_0011;
      L     0; // number additional param
      T     "SSA_LOG_Value_Queue".Input.Para_0012;
// cont log-messages
      L     "SSA_LOG_Value_Queue".Input.Para_0099; // message counter
      L     1;
      +I    ;
      T     "SSA_LOG_Value_Queue".Input.Para_0099; // message counter

// Transform Basic Time to Local Time
//      CALL  "BT_LT"
//       BT     :="DB Prozesszeit".Arbeitsbereich.dt1
//       WS_DAT :="RegelDB"
//       RET_VAL:=MW218
//       LT     :="RegelDB".LocalTime
// put timestamp into message
      CALL "SYS_Copy_DBtoDB" (
           DBSource                 := 1013,
           ByteSource               := 18,
           DBDest                   := 1005,
           ByteDest                 := 462,
           NoOfByte                 := 8,
           Fault                    := M    210.0);
///
      CALL "SSA_MH_LogEntry_ActValue" (
           DBNumber                 := 1005);

E084: NOP   0;
///
// Ereignis 38  Kommt
      U     #EREIGNISBIT_38;
      FP    #Ereignis_38.FP_Kommt;
      SPBN  E085;
// header
      L     #MessageType;
      T     "SSA_LOG_Value_Queue".Input.Header.SecType; // type
      L     #MessageFormat;
      T     "SSA_LOG_Value_Queue".Input.Header.Format; // format
      L     #JobNumber;
      T     "SSA_LOG_Value_Queue".Input.Para_0005;
      L     #processMinute;
      T     "SSA_LOG_Value_Queue".Input.Para_0007;
      L     #StepNumber;
      T     "SSA_LOG_Value_Queue".Input.Para_0008;
      L     #StepTimeMin;
      T     "SSA_LOG_Value_Queue".Input.Para_0009;

// values integer
      L     #EventObject_38; // event-Nr
      T     "SSA_LOG_Value_Queue".Input.Para_0010;
      L     1; // object-state coming
      T     "SSA_LOG_Value_Queue".Input.Para_0011;
      L     0; // number additional param
      T     "SSA_LOG_Value_Queue".Input.Para_0012;
// cont log-messages
      L     "SSA_LOG_Value_Queue".Input.Para_0099; // message counter
      L     1;
      +I    ;
      T     "SSA_LOG_Value_Queue".Input.Para_0099; // message counter

// Transform Basic Time to Local Time
//      CALL  "BT_LT"
//       BT     :="DB Prozesszeit".Arbeitsbereich.dt1
//       WS_DAT :="RegelDB"
//       RET_VAL:=MW218
//       LT     :="RegelDB".LocalTime
// put timestamp into message
      CALL "SYS_Copy_DBtoDB" (
           DBSource                 := 1013,
           ByteSource               := 18,
           DBDest                   := 1005,
           ByteDest                 := 462,
           NoOfByte                 := 8,
           Fault                    := M    210.0);
///
      CALL "SSA_MH_LogEntry_ActValue" (
           DBNumber                 := 1005);

E085: NOP   0;
///
// Ereignis 38  Geht
      U     #EREIGNISBIT_38;
      FN    #Ereignis_38.FN_Geht;
      SPBN  E086;
// header
      L     #MessageType;
      T     "SSA_LOG_Value_Queue".Input.Header.SecType; // type
      L     #MessageFormat;
      T     "SSA_LOG_Value_Queue".Input.Header.Format; // format
      L     #JobNumber;
      T     "SSA_LOG_Value_Queue".Input.Para_0005;
      L     #processMinute;
      T     "SSA_LOG_Value_Queue".Input.Para_0007;
      L     #StepNumber;
      T     "SSA_LOG_Value_Queue".Input.Para_0008;
      L     #StepTimeMin;
      T     "SSA_LOG_Value_Queue".Input.Para_0009;

// values integer
      L     #EventObject_38; // event-Nr
      T     "SSA_LOG_Value_Queue".Input.Para_0010;
      L     2; // object-state going
      T     "SSA_LOG_Value_Queue".Input.Para_0011;
      L     0; // number additional param
      T     "SSA_LOG_Value_Queue".Input.Para_0012;
// cont log-messages
      L     "SSA_LOG_Value_Queue".Input.Para_0099; // message counter
      L     1;
      +I    ;
      T     "SSA_LOG_Value_Queue".Input.Para_0099; // message counter

// Transform Basic Time to Local Time
//      CALL  "BT_LT"
//       BT     :="DB Prozesszeit".Arbeitsbereich.dt1
//       WS_DAT :="RegelDB"
//       RET_VAL:=MW218
//       LT     :="RegelDB".LocalTime
// put timestamp into message
      CALL "SYS_Copy_DBtoDB" (
           DBSource                 := 1013,
           ByteSource               := 18,
           DBDest                   := 1005,
           ByteDest                 := 462,
           NoOfByte                 := 8,
           Fault                    := M    210.0);
///
      CALL "SSA_MH_LogEntry_ActValue" (
           DBNumber                 := 1005);

E086: NOP   0;
///
// Ereignis 39  Kommt
      U     #EREIGNISBIT_39;
      FP    #Ereignis_39.FP_Kommt;
      SPBN  E087;
// header
      L     #MessageType;
      T     "SSA_LOG_Value_Queue".Input.Header.SecType; // type
      L     #MessageFormat;
      T     "SSA_LOG_Value_Queue".Input.Header.Format; // format
      L     #JobNumber;
      T     "SSA_LOG_Value_Queue".Input.Para_0005;
      L     #processMinute;
      T     "SSA_LOG_Value_Queue".Input.Para_0007;
      L     #StepNumber;
      T     "SSA_LOG_Value_Queue".Input.Para_0008;
      L     #StepTimeMin;
      T     "SSA_LOG_Value_Queue".Input.Para_0009;

// values integer
      L     #EventObject_39; // event-Nr
      T     "SSA_LOG_Value_Queue".Input.Para_0010;
      L     1; // object-state coming
      T     "SSA_LOG_Value_Queue".Input.Para_0011;
      L     0; // number additional param
      T     "SSA_LOG_Value_Queue".Input.Para_0012;
// cont log-messages
      L     "SSA_LOG_Value_Queue".Input.Para_0099; // message counter
      L     1;
      +I    ;
      T     "SSA_LOG_Value_Queue".Input.Para_0099; // message counter

// Transform Basic Time to Local Time
//      CALL  "BT_LT"
//       BT     :="DB Prozesszeit".Arbeitsbereich.dt1
//       WS_DAT :="RegelDB"
//       RET_VAL:=MW218
//       LT     :="RegelDB".LocalTime
// put timestamp into message
      CALL "SYS_Copy_DBtoDB" (
           DBSource                 := 1013,
           ByteSource               := 18,
           DBDest                   := 1005,
           ByteDest                 := 462,
           NoOfByte                 := 8,
           Fault                    := M    210.0);
///
      CALL "SSA_MH_LogEntry_ActValue" (
           DBNumber                 := 1005);

E087: NOP   0;
///
// Ereignis 39  Geht
      U     #EREIGNISBIT_39;
      FN    #Ereignis_39.FN_Geht;
      SPBN  E088;
// header
      L     #MessageType;
      T     "SSA_LOG_Value_Queue".Input.Header.SecType; // type
      L     #MessageFormat;
      T     "SSA_LOG_Value_Queue".Input.Header.Format; // format
      L     #JobNumber;
      T     "SSA_LOG_Value_Queue".Input.Para_0005;
      L     #processMinute;
      T     "SSA_LOG_Value_Queue".Input.Para_0007;
      L     #StepNumber;
      T     "SSA_LOG_Value_Queue".Input.Para_0008;
      L     #StepTimeMin;
      T     "SSA_LOG_Value_Queue".Input.Para_0009;

// values integer
      L     #EventObject_39; // event-Nr
      T     "SSA_LOG_Value_Queue".Input.Para_0010;
      L     2; // object-state going
      T     "SSA_LOG_Value_Queue".Input.Para_0011;
      L     0; // number additional param
      T     "SSA_LOG_Value_Queue".Input.Para_0012;
// cont log-messages
      L     "SSA_LOG_Value_Queue".Input.Para_0099; // message counter
      L     1;
      +I    ;
      T     "SSA_LOG_Value_Queue".Input.Para_0099; // message counter

// Transform Basic Time to Local Time
//      CALL  "BT_LT"
//       BT     :="DB Prozesszeit".Arbeitsbereich.dt1
//       WS_DAT :="RegelDB"
//       RET_VAL:=MW218
//       LT     :="RegelDB".LocalTime
// put timestamp into message
      CALL "SYS_Copy_DBtoDB" (
           DBSource                 := 1013,
           ByteSource               := 18,
           DBDest                   := 1005,
           ByteDest                 := 462,
           NoOfByte                 := 8,
           Fault                    := M    210.0);
///
      CALL "SSA_MH_LogEntry_ActValue" (
           DBNumber                 := 1005);

E088: NOP   0;
///
// Ereignis 40  Kommt
      U     #EREIGNISBIT_40;
      FP    #Ereignis_40.FP_Kommt;
      SPBN  E089;
// header
      L     #MessageType;
      T     "SSA_LOG_Value_Queue".Input.Header.SecType; // type
      L     #MessageFormat;
      T     "SSA_LOG_Value_Queue".Input.Header.Format; // format
      L     #JobNumber;
      T     "SSA_LOG_Value_Queue".Input.Para_0005;
      L     #processMinute;
      T     "SSA_LOG_Value_Queue".Input.Para_0007;
      L     #StepNumber;
      T     "SSA_LOG_Value_Queue".Input.Para_0008;
      L     #StepTimeMin;
      T     "SSA_LOG_Value_Queue".Input.Para_0009;

// values integer
      L     #EventObject_40; // event-Nr
      T     "SSA_LOG_Value_Queue".Input.Para_0010;
      L     1; // object-state coming
      T     "SSA_LOG_Value_Queue".Input.Para_0011;
      L     0; // number additional param
      T     "SSA_LOG_Value_Queue".Input.Para_0012;
// cont log-messages
      L     "SSA_LOG_Value_Queue".Input.Para_0099; // message counter
      L     1;
      +I    ;
      T     "SSA_LOG_Value_Queue".Input.Para_0099; // message counter

// Transform Basic Time to Local Time
//      CALL  "BT_LT"
//       BT     :="DB Prozesszeit".Arbeitsbereich.dt1
//       WS_DAT :="RegelDB"
//       RET_VAL:=MW218
//       LT     :="RegelDB".LocalTime
// put timestamp into message
      CALL "SYS_Copy_DBtoDB" (
           DBSource                 := 1013,
           ByteSource               := 18,
           DBDest                   := 1005,
           ByteDest                 := 462,
           NoOfByte                 := 8,
           Fault                    := M    210.0);
///
      CALL "SSA_MH_LogEntry_ActValue" (
           DBNumber                 := 1005);

E089: NOP   0;
///
// Ereignis 40  Geht
      U     #EREIGNISBIT_40;
      FN    #Ereignis_40.FN_Geht;
      SPBN  E090;
// header
      L     #MessageType;
      T     "SSA_LOG_Value_Queue".Input.Header.SecType; // type
      L     #MessageFormat;
      T     "SSA_LOG_Value_Queue".Input.Header.Format; // format
      L     #JobNumber;
      T     "SSA_LOG_Value_Queue".Input.Para_0005;
      L     #processMinute;
      T     "SSA_LOG_Value_Queue".Input.Para_0007;
      L     #StepNumber;
      T     "SSA_LOG_Value_Queue".Input.Para_0008;
      L     #StepTimeMin;
      T     "SSA_LOG_Value_Queue".Input.Para_0009;

// values integer
      L     #EventObject_40; // event-Nr
      T     "SSA_LOG_Value_Queue".Input.Para_0010;
      L     2; // object-state going
      T     "SSA_LOG_Value_Queue".Input.Para_0011;
      L     0; // number additional param
      T     "SSA_LOG_Value_Queue".Input.Para_0012;
// cont log-messages
      L     "SSA_LOG_Value_Queue".Input.Para_0099; // message counter
      L     1;
      +I    ;
      T     "SSA_LOG_Value_Queue".Input.Para_0099; // message counter

// Transform Basic Time to Local Time
//      CALL  "BT_LT"
//       BT     :="DB Prozesszeit".Arbeitsbereich.dt1
//       WS_DAT :="RegelDB"
//       RET_VAL:=MW218
//       LT     :="RegelDB".LocalTime
// put timestamp into message
      CALL "SYS_Copy_DBtoDB" (
           DBSource                 := 1013,
           ByteSource               := 18,
           DBDest                   := 1005,
           ByteDest                 := 462,
           NoOfByte                 := 8,
           Fault                    := M    210.0);
///
      CALL "SSA_MH_LogEntry_ActValue" (
           DBNumber                 := 1005);

E090: NOP   0;
///
// Ereignis 41  Kommt
      U     #EREIGNISBIT_41;
      FP    #Ereignis_41.FP_Kommt;
      SPBN  E091;
// header
      L     #MessageType;
      T     "SSA_LOG_Value_Queue".Input.Header.SecType; // type
      L     #MessageFormat;
      T     "SSA_LOG_Value_Queue".Input.Header.Format; // format
      L     #JobNumber;
      T     "SSA_LOG_Value_Queue".Input.Para_0005;
      L     #processMinute;
      T     "SSA_LOG_Value_Queue".Input.Para_0007;
      L     #StepNumber;
      T     "SSA_LOG_Value_Queue".Input.Para_0008;
      L     #StepTimeMin;
      T     "SSA_LOG_Value_Queue".Input.Para_0009;

// values integer
      L     #EventObject_41; // event-Nr
      T     "SSA_LOG_Value_Queue".Input.Para_0010;
      L     1; // object-state coming
      T     "SSA_LOG_Value_Queue".Input.Para_0011;
      L     0; // number additional param
      T     "SSA_LOG_Value_Queue".Input.Para_0012;
// cont log-messages
      L     "SSA_LOG_Value_Queue".Input.Para_0099; // message counter
      L     1;
      +I    ;
      T     "SSA_LOG_Value_Queue".Input.Para_0099; // message counter

// Transform Basic Time to Local Time
//      CALL  "BT_LT"
//       BT     :="DB Prozesszeit".Arbeitsbereich.dt1
//       WS_DAT :="RegelDB"
//       RET_VAL:=MW218
//       LT     :="RegelDB".LocalTime
// put timestamp into message
      CALL "SYS_Copy_DBtoDB" (
           DBSource                 := 1013,
           ByteSource               := 18,
           DBDest                   := 1005,
           ByteDest                 := 462,
           NoOfByte                 := 8,
           Fault                    := M    210.0);
///
      CALL "SSA_MH_LogEntry_ActValue" (
           DBNumber                 := 1005);

E091: NOP   0;
///
// Ereignis 41  Geht
      U     #EREIGNISBIT_41;
      FN    #Ereignis_41.FN_Geht;
      SPBN  E092;
// header
      L     #MessageType;
      T     "SSA_LOG_Value_Queue".Input.Header.SecType; // type
      L     #MessageFormat;
      T     "SSA_LOG_Value_Queue".Input.Header.Format; // format
      L     #JobNumber;
      T     "SSA_LOG_Value_Queue".Input.Para_0005;
      L     #processMinute;
      T     "SSA_LOG_Value_Queue".Input.Para_0007;
      L     #StepNumber;
      T     "SSA_LOG_Value_Queue".Input.Para_0008;
      L     #StepTimeMin;
      T     "SSA_LOG_Value_Queue".Input.Para_0009;

// values integer
      L     #EventObject_41; // event-Nr
      T     "SSA_LOG_Value_Queue".Input.Para_0010;
      L     2; // object-state going
      T     "SSA_LOG_Value_Queue".Input.Para_0011;
      L     0; // number additional param
      T     "SSA_LOG_Value_Queue".Input.Para_0012;
// cont log-messages
      L     "SSA_LOG_Value_Queue".Input.Para_0099; // message counter
      L     1;
      +I    ;
      T     "SSA_LOG_Value_Queue".Input.Para_0099; // message counter

// Transform Basic Time to Local Time
//      CALL  "BT_LT"
//       BT     :="DB Prozesszeit".Arbeitsbereich.dt1
//       WS_DAT :="RegelDB"
//       RET_VAL:=MW218
//       LT     :="RegelDB".LocalTime
// put timestamp into message
      CALL "SYS_Copy_DBtoDB" (
           DBSource                 := 1013,
           ByteSource               := 18,
           DBDest                   := 1005,
           ByteDest                 := 462,
           NoOfByte                 := 8,
           Fault                    := M    210.0);
///
      CALL "SSA_MH_LogEntry_ActValue" (
           DBNumber                 := 1005);

E092: NOP   0;
///
// Ereignis 42  Kommt
      U     #EREIGNISBIT_42;
      FP    #Ereignis_42.FP_Kommt;
      SPBN  E093;
// header
      L     #MessageType;
      T     "SSA_LOG_Value_Queue".Input.Header.SecType; // type
      L     #MessageFormat;
      T     "SSA_LOG_Value_Queue".Input.Header.Format; // format
      L     #JobNumber;
      T     "SSA_LOG_Value_Queue".Input.Para_0005;
      L     #processMinute;
      T     "SSA_LOG_Value_Queue".Input.Para_0007;
      L     #StepNumber;
      T     "SSA_LOG_Value_Queue".Input.Para_0008;
      L     #StepTimeMin;
      T     "SSA_LOG_Value_Queue".Input.Para_0009;

// values integer
      L     #EventObject_42; // event-Nr
      T     "SSA_LOG_Value_Queue".Input.Para_0010;
      L     1; // object-state coming
      T     "SSA_LOG_Value_Queue".Input.Para_0011;
      L     0; // number additional param
      T     "SSA_LOG_Value_Queue".Input.Para_0012;
// cont log-messages
      L     "SSA_LOG_Value_Queue".Input.Para_0099; // message counter
      L     1;
      +I    ;
      T     "SSA_LOG_Value_Queue".Input.Para_0099; // message counter

// Transform Basic Time to Local Time
//      CALL  "BT_LT"
//       BT     :="DB Prozesszeit".Arbeitsbereich.dt1
//       WS_DAT :="RegelDB"
//       RET_VAL:=MW218
//       LT     :="RegelDB".LocalTime
// put timestamp into message
      CALL "SYS_Copy_DBtoDB" (
           DBSource                 := 1013,
           ByteSource               := 18,
           DBDest                   := 1005,
           ByteDest                 := 462,
           NoOfByte                 := 8,
           Fault                    := M    210.0);
///
      CALL "SSA_MH_LogEntry_ActValue" (
           DBNumber                 := 1005);

E093: NOP   0;
///
// Ereignis 42  Geht
      U     #EREIGNISBIT_42;
      FN    #Ereignis_42.FN_Geht;
      SPBN  E094;
// header
      L     #MessageType;
      T     "SSA_LOG_Value_Queue".Input.Header.SecType; // type
      L     #MessageFormat;
      T     "SSA_LOG_Value_Queue".Input.Header.Format; // format
      L     #JobNumber;
      T     "SSA_LOG_Value_Queue".Input.Para_0005;
      L     #processMinute;
      T     "SSA_LOG_Value_Queue".Input.Para_0007;
      L     #StepNumber;
      T     "SSA_LOG_Value_Queue".Input.Para_0008;
      L     #StepTimeMin;
      T     "SSA_LOG_Value_Queue".Input.Para_0009;

// values integer
      L     #EventObject_42; // event-Nr
      T     "SSA_LOG_Value_Queue".Input.Para_0010;
      L     2; // object-state going
      T     "SSA_LOG_Value_Queue".Input.Para_0011;
      L     0; // number additional param
      T     "SSA_LOG_Value_Queue".Input.Para_0012;
// cont log-messages
      L     "SSA_LOG_Value_Queue".Input.Para_0099; // message counter
      L     1;
      +I    ;
      T     "SSA_LOG_Value_Queue".Input.Para_0099; // message counter

// Transform Basic Time to Local Time
//      CALL  "BT_LT"
//       BT     :="DB Prozesszeit".Arbeitsbereich.dt1
//       WS_DAT :="RegelDB"
//       RET_VAL:=MW218
//       LT     :="RegelDB".LocalTime
// put timestamp into message
      CALL "SYS_Copy_DBtoDB" (
           DBSource                 := 1013,
           ByteSource               := 18,
           DBDest                   := 1005,
           ByteDest                 := 462,
           NoOfByte                 := 8,
           Fault                    := M    210.0);
///
      CALL "SSA_MH_LogEntry_ActValue" (
           DBNumber                 := 1005);

E094: NOP   0;
///
// Ereignis 43  Kommt
      U     #EREIGNISBIT_43;
      FP    #Ereignis_43.FP_Kommt;
      SPBN  E095;
// header
      L     #MessageType;
      T     "SSA_LOG_Value_Queue".Input.Header.SecType; // type
      L     #MessageFormat;
      T     "SSA_LOG_Value_Queue".Input.Header.Format; // format
      L     #JobNumber;
      T     "SSA_LOG_Value_Queue".Input.Para_0005;
      L     #processMinute;
      T     "SSA_LOG_Value_Queue".Input.Para_0007;
      L     #StepNumber;
      T     "SSA_LOG_Value_Queue".Input.Para_0008;
      L     #StepTimeMin;
      T     "SSA_LOG_Value_Queue".Input.Para_0009;

// values integer
      L     #EventObject_43; // event-Nr
      T     "SSA_LOG_Value_Queue".Input.Para_0010;
      L     1; // object-state coming
      T     "SSA_LOG_Value_Queue".Input.Para_0011;
      L     0; // number additional param
      T     "SSA_LOG_Value_Queue".Input.Para_0012;
// cont log-messages
      L     "SSA_LOG_Value_Queue".Input.Para_0099; // message counter
      L     1;
      +I    ;
      T     "SSA_LOG_Value_Queue".Input.Para_0099; // message counter

// Transform Basic Time to Local Time
//      CALL  "BT_LT"
//       BT     :="DB Prozesszeit".Arbeitsbereich.dt1
//       WS_DAT :="RegelDB"
//       RET_VAL:=MW218
//       LT     :="RegelDB".LocalTime
// put timestamp into message
      CALL "SYS_Copy_DBtoDB" (
           DBSource                 := 1013,
           ByteSource               := 18,
           DBDest                   := 1005,
           ByteDest                 := 462,
           NoOfByte                 := 8,
           Fault                    := M    210.0);
///
      CALL "SSA_MH_LogEntry_ActValue" (
           DBNumber                 := 1005);

E095: NOP   0;
///
// Ereignis 43  Geht
      U     #EREIGNISBIT_43;
      FN    #Ereignis_43.FN_Geht;
      SPBN  E096;
// header
      L     #MessageType;
      T     "SSA_LOG_Value_Queue".Input.Header.SecType; // type
      L     #MessageFormat;
      T     "SSA_LOG_Value_Queue".Input.Header.Format; // format
      L     #JobNumber;
      T     "SSA_LOG_Value_Queue".Input.Para_0005;
      L     #processMinute;
      T     "SSA_LOG_Value_Queue".Input.Para_0007;
      L     #StepNumber;
      T     "SSA_LOG_Value_Queue".Input.Para_0008;
      L     #StepTimeMin;
      T     "SSA_LOG_Value_Queue".Input.Para_0009;

// values integer
      L     #EventObject_43; // event-Nr
      T     "SSA_LOG_Value_Queue".Input.Para_0010;
      L     2; // object-state going
      T     "SSA_LOG_Value_Queue".Input.Para_0011;
      L     0; // number additional param
      T     "SSA_LOG_Value_Queue".Input.Para_0012;
// cont log-messages
      L     "SSA_LOG_Value_Queue".Input.Para_0099; // message counter
      L     1;
      +I    ;
      T     "SSA_LOG_Value_Queue".Input.Para_0099; // message counter

// Transform Basic Time to Local Time
//      CALL  "BT_LT"
//       BT     :="DB Prozesszeit".Arbeitsbereich.dt1
//       WS_DAT :="RegelDB"
//       RET_VAL:=MW218
//       LT     :="RegelDB".LocalTime
// put timestamp into message
      CALL "SYS_Copy_DBtoDB" (
           DBSource                 := 1013,
           ByteSource               := 18,
           DBDest                   := 1005,
           ByteDest                 := 462,
           NoOfByte                 := 8,
           Fault                    := M    210.0);
///
      CALL "SSA_MH_LogEntry_ActValue" (
           DBNumber                 := 1005);

E096: NOP   0;
///
// Ereignis 44  Kommt
      U     #EREIGNISBIT_44;
      FP    #Ereignis_44.HP_Kommt;
      SPBN  E097;
// header
      L     #MessageType;
      T     "SSA_LOG_Value_Queue".Input.Header.SecType; // type
      L     #MessageFormat;
      T     "SSA_LOG_Value_Queue".Input.Header.Format; // format
      L     #JobNumber;
      T     "SSA_LOG_Value_Queue".Input.Para_0005;
      L     #processMinute;
      T     "SSA_LOG_Value_Queue".Input.Para_0007;
      L     #StepNumber;
      T     "SSA_LOG_Value_Queue".Input.Para_0008;
      L     #StepTimeMin;
      T     "SSA_LOG_Value_Queue".Input.Para_0009;

// values integer
      L     #EventObject_44; // event-Nr
      T     "SSA_LOG_Value_Queue".Input.Para_0010;
      L     1; // object-state coming
      T     "SSA_LOG_Value_Queue".Input.Para_0011;
      L     0; // number additional param
      T     "SSA_LOG_Value_Queue".Input.Para_0012;
// cont log-messages
      L     "SSA_LOG_Value_Queue".Input.Para_0099; // message counter
      L     1;
      +I    ;
      T     "SSA_LOG_Value_Queue".Input.Para_0099; // message counter

// Transform Basic Time to Local Time
//      CALL  "BT_LT"
//       BT     :="DB Prozesszeit".Arbeitsbereich.dt1
//       WS_DAT :="RegelDB"
//       RET_VAL:=MW218
//       LT     :="RegelDB".LocalTime
// put timestamp into message
      CALL "SYS_Copy_DBtoDB" (
           DBSource                 := 1013,
           ByteSource               := 18,
           DBDest                   := 1005,
           ByteDest                 := 462,
           NoOfByte                 := 8,
           Fault                    := M    210.0);
///
      CALL "SSA_MH_LogEntry_ActValue" (
           DBNumber                 := 1005);

E097: NOP   0;
///
// Ereignis 44  Geht
      U     #EREIGNISBIT_44;
      FN    #Ereignis_44.HP_Geht;
      SPBN  E098;
// header
      L     #MessageType;
      T     "SSA_LOG_Value_Queue".Input.Header.SecType; // type
      L     #MessageFormat;
      T     "SSA_LOG_Value_Queue".Input.Header.Format; // format
      L     #JobNumber;
      T     "SSA_LOG_Value_Queue".Input.Para_0005;
      L     #processMinute;
      T     "SSA_LOG_Value_Queue".Input.Para_0007;
      L     #StepNumber;
      T     "SSA_LOG_Value_Queue".Input.Para_0008;
      L     #StepTimeMin;
      T     "SSA_LOG_Value_Queue".Input.Para_0009;

// values integer
      L     #EventObject_44; // event-Nr
      T     "SSA_LOG_Value_Queue".Input.Para_0010;
      L     2; // object-state going
      T     "SSA_LOG_Value_Queue".Input.Para_0011;
      L     0; // number additional param
      T     "SSA_LOG_Value_Queue".Input.Para_0012;
// cont log-messages
      L     "SSA_LOG_Value_Queue".Input.Para_0099; // message counter
      L     1;
      +I    ;
      T     "SSA_LOG_Value_Queue".Input.Para_0099; // message counter

// Transform Basic Time to Local Time
//      CALL  "BT_LT"
//       BT     :="DB Prozesszeit".Arbeitsbereich.dt1
//       WS_DAT :="RegelDB"
//       RET_VAL:=MW218
//       LT     :="RegelDB".LocalTime
// put timestamp into message
      CALL "SYS_Copy_DBtoDB" (
           DBSource                 := 1013,
           ByteSource               := 18,
           DBDest                   := 1005,
           ByteDest                 := 462,
           NoOfByte                 := 8,
           Fault                    := M    210.0);
///
      CALL "SSA_MH_LogEntry_ActValue" (
           DBNumber                 := 1005);

E098: NOP   0;

NETWORK
TITLE =



NETWORK
TITLE =Test-Event
// Ereignis 47 Kommt
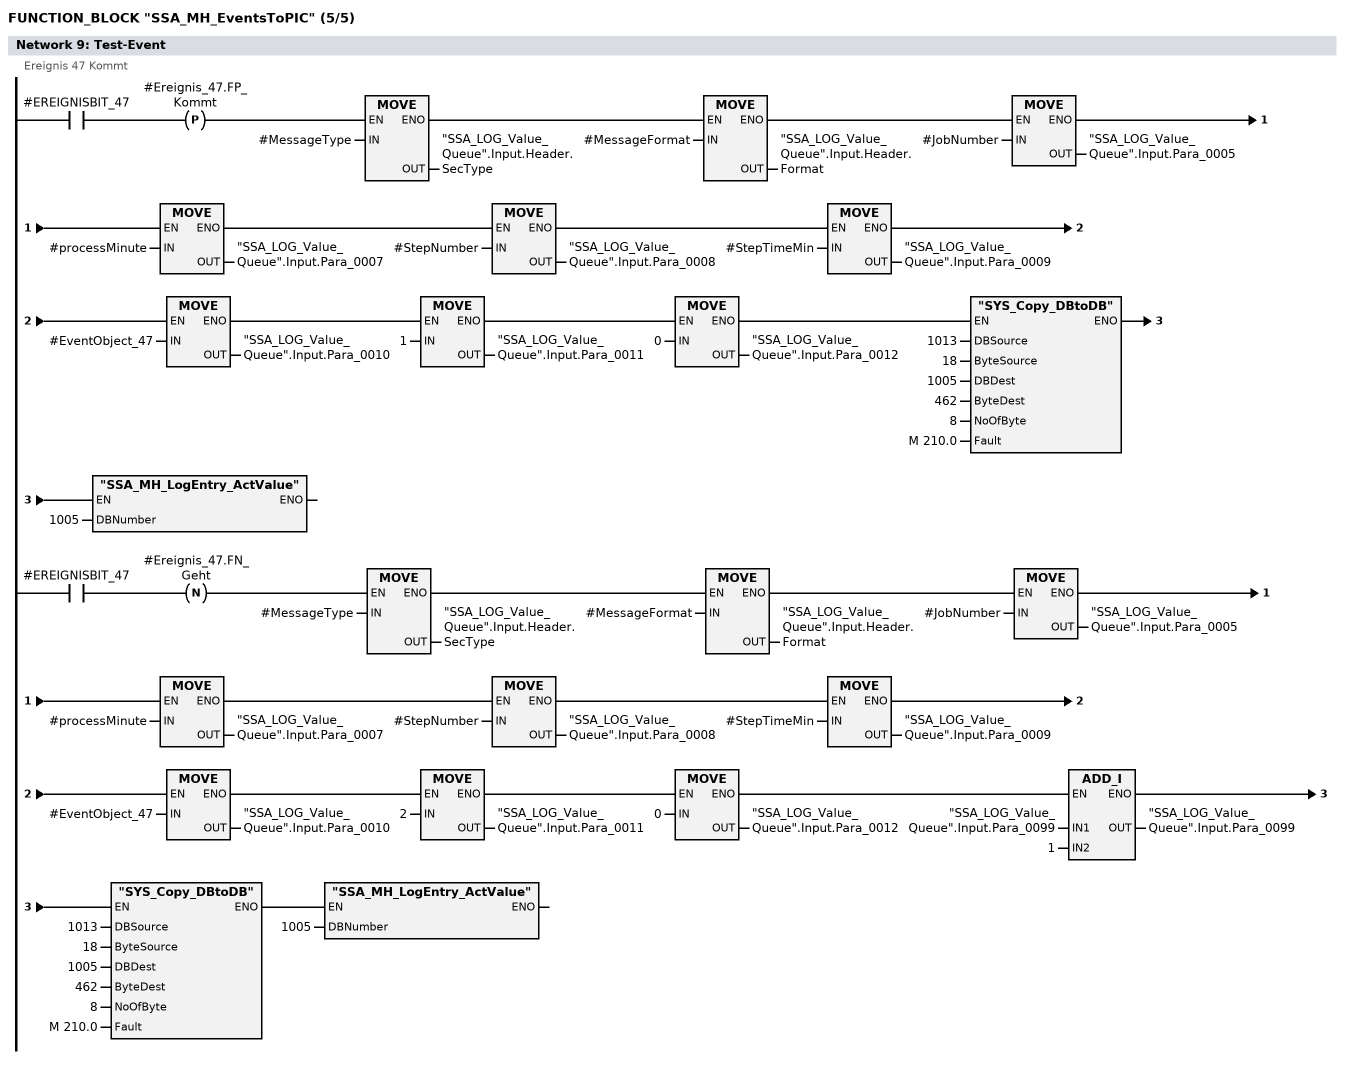
      U     #EREIGNISBIT_47;
      FP    #Ereignis_47.FP_Kommt;
      SPBN  E993;
// header
      L     #MessageType;
      T     "SSA_LOG_Value_Queue".Input.Header.SecType; // type
      L     #MessageFormat;
      T     "SSA_LOG_Value_Queue".Input.Header.Format; // format
      L     #JobNumber;
      T     "SSA_LOG_Value_Queue".Input.Para_0005;
      L     #processMinute;
      T     "SSA_LOG_Value_Queue".Input.Para_0007;
      L     #StepNumber;
      T     "SSA_LOG_Value_Queue".Input.Para_0008;
      L     #StepTimeMin;
      T     "SSA_LOG_Value_Queue".Input.Para_0009;

// values integer
      L     #EventObject_47; // event-Nr
      T     "SSA_LOG_Value_Queue".Input.Para_0010;
      L     1; // object-state coming
      T     "SSA_LOG_Value_Queue".Input.Para_0011;
      L     0; // number additional param
      T     "SSA_LOG_Value_Queue".Input.Para_0012;

//      CALL  "BT_LT"
//       BT     :="DB Prozesszeit".Arbeitsbereich.dt1
//       WS_DAT :="RegelDB"
//       RET_VAL:=MW218
//       LT     :="RegelDB".LocalTime
      CALL "SYS_Copy_DBtoDB" (
           DBSource                 := 1013,
           ByteSource               := 18,
           DBDest                   := 1005,
           ByteDest                 := 462,
           NoOfByte                 := 8,
           Fault                    := M    210.0);
      CALL "SSA_MH_LogEntry_ActValue" (
           DBNumber                 := 1005);
E993: NOP   0;

// Ereignis 47 Geht
      U     #EREIGNISBIT_47;
      FN    #Ereignis_47.FN_Geht;
      SPBN  E994;
// header
      L     #MessageType;
      T     "SSA_LOG_Value_Queue".Input.Header.SecType; // type
      L     #MessageFormat;
      T     "SSA_LOG_Value_Queue".Input.Header.Format; // format
      L     #JobNumber;
      T     "SSA_LOG_Value_Queue".Input.Para_0005;
      L     #processMinute;
      T     "SSA_LOG_Value_Queue".Input.Para_0007;
      L     #StepNumber;
      T     "SSA_LOG_Value_Queue".Input.Para_0008;
      L     #StepTimeMin;
      T     "SSA_LOG_Value_Queue".Input.Para_0009;

// values integer
      L     #EventObject_47; // event-Nr
      T     "SSA_LOG_Value_Queue".Input.Para_0010;
      L     2; // object-state going
      T     "SSA_LOG_Value_Queue".Input.Para_0011;
      L     0; // number additional param
      T     "SSA_LOG_Value_Queue".Input.Para_0012;
// cont log-messages
      L     "SSA_LOG_Value_Queue".Input.Para_0099; // message counter
      L     1;
      +I    ;
      T     "SSA_LOG_Value_Queue".Input.Para_0099; // message counter

//      CALL  "BT_LT"
//       BT     :="DB Prozesszeit".Arbeitsbereich.dt1
//       WS_DAT :="RegelDB"
//       RET_VAL:=MW218
//       LT     :="RegelDB".LocalTime
      CALL "SYS_Copy_DBtoDB" (
           DBSource                 := 1013,
           ByteSource               := 18,
           DBDest                   := 1005,
           ByteDest                 := 462,
           NoOfByte                 := 8,
           Fault                    := M    210.0);

      CALL "SSA_MH_LogEntry_ActValue" (
           DBNumber                 := 1005);
E994: NOP   0;


NETWORK
TITLE =
//Blinker zum testen
      UN    T     29;

      L     S5T#2S;
      SE    T     28;
      U     T     28;
      L     S5T#2S;
      SE    T     29;
      CLR   ;
      =     M    300.0;

NETWORK
TITLE =

      BE    ;

END_FUNCTION_BLOCK

